# EPICS autosave request: gardasoftLED/PP420Profile_settings.req
$(P):PR$(PROFILE):MODE
$(P):PR$(PROFILE):NAME
